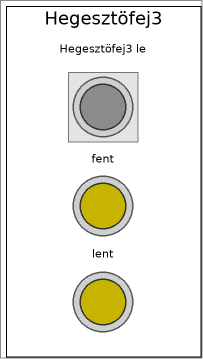
VISUALIZATION Hegesztofej_IOk_Pt  // 203x359
    Rectangle (6,6 195x351), "Hegesztöfej3"
    Lamp1 (68,171 70x70), variable: GVL.bHegeszto3Fent, style: Lamp-Lamp1-Yellow
    Label (73,149 60x20), "fent"
    Lamp1 (68,267 70x70), variable: GVL.bHegeszto3Lent, style: Lamp-Lamp1-Yellow
    Label (73,244 60x20), "lent"
    Label (45,39 116x20), "Hegesztöfej3 le"
    PushSwitch (68,72 70x70), variable: HEGESZTOK.bHegesztoFejekOutput[2], behaviour: TOGGLE, style: Switch-PushSwitch-Gray
END_VISUALIZATION

(* stored: Version 1.1.0.1, ProductVersion 3.1.4024.11
   Visu Hegesztofej_IOk_Pt: Id {fb7815da-7e04-4a5c-8edc-27a3ec4bda53} *)
